  MoveL 11412 to (239.47, 155.25, 153.89) mm, rotated rx 180 ry 0 rz -180 deg; joints [-62.893, 69.046, -92.108, 64.781, 100.282, 20.756]
  MoveL 11413 to (239.47, 155.25, 153.89) mm, rotated rx 180 ry 0 rz -180 deg; joints [-62.893, 69.046, -92.108, 64.781, 100.282, 20.756]
  Call Extruder(262.89466)
  MoveL 11414 to (239.41, 155.44, 153.89) mm, rotated rx 180 ry 0 rz -180 deg; joints [-62.939, 69.059, -92.103, 64.822, 100.258, 20.747]
  MoveL 11415 to (239.41, 155.44, 153.89) mm, rotated rx 180 ry 0 rz -180 deg; joints [-62.939, 69.059, -92.103, 64.822, 100.258, 20.747]
  Call Extruder(263.07662)
  MoveL 11416 to (239.29, 155.73, 153.89) mm, rotated rx 180 ry 0 rz 180 deg; joints [-63.018, 69.079, -92.095, 64.892, 100.218, 20.735]
  MoveL 11417 to (239.29, 155.73, 153.89) mm, rotated rx 180 ry 0 rz 180 deg; joints [-63.018, 69.079, -92.095, 64.892, 100.218, 20.735]
  Call Extruder(263.25933)
  MoveL 11418 to (239.17, 156.02, 153.89) mm, rotated rx 180 ry 0 rz 180 deg; joints [-63.097, 69.098, -92.087, 64.963, 100.179, 20.723]
  MoveL 11419 to (239.17, 156.02, 153.89) mm, rotated rx 180 ry 0 rz 180 deg; joints [-63.097, 69.098, -92.087, 64.963, 100.179, 20.723]
  Call Extruder(263.42975)
  MoveL 11420 to (239.05, 156.29, 153.89) mm, rotated rx 180 ry 0 rz 180 deg; joints [-63.17, 69.116, -92.079, 65.028, 100.142, 20.712]
  MoveL 11421 to (239.05, 156.29, 153.89) mm, rotated rx 180 ry 0 rz 180 deg; joints [-63.17, 69.116, -92.079, 65.028, 100.142, 20.712]
  Call Extruder(263.58776)
  MoveL 11422 to (238.94, 156.54, 153.89) mm, rotated rx 180 ry 0 rz 180 deg; joints [-63.238, 69.132, -92.073, 65.089, 100.108, 20.702]
  MoveL 11423 to (238.94, 156.54, 153.89) mm, rotated rx 180 ry 0 rz 180 deg; joints [-63.238, 69.132, -92.073, 65.089, 100.108, 20.702]
  Call Extruder(263.74638)
  MoveL 11424 to (238.84, 156.79, 153.89) mm, rotated rx 180 ry 0 rz -180 deg; joints [-63.306, 69.149, -92.066, 65.15, 100.074, 20.692]
  MoveL 11425 to (238.84, 156.79, 153.89) mm, rotated rx 180 ry 0 rz -180 deg; joints [-63.306, 69.149, -92.066, 65.15, 100.074, 20.692]
  Call Extruder(263.95255)
  MoveL 11426 to (238.66, 157.09, 153.89) mm, rotated rx 180 ry 0 rz 180 deg; joints [-63.401, 69.167, -92.058, 65.236, 100.03, 20.684]
  MoveL 11427 to (238.66, 157.09, 153.89) mm, rotated rx 180 ry 0 rz 180 deg; joints [-63.401, 69.167, -92.058, 65.236, 100.03, 20.684]
  Call Extruder(264.15949)
  MoveL 11428 to (238.49, 157.4, 153.89) mm, rotated rx 180 ry 0 rz 180 deg; joints [-63.497, 69.185, -92.05, 65.323, 99.985, 20.676]
  MoveL 11429 to (238.49, 157.4, 153.89) mm, rotated rx 180 ry 0 rz 180 deg; joints [-63.497, 69.185, -92.05, 65.323, 99.985, 20.676]
  Call Extruder(264.36722)
  MoveL 11430 to (238.31, 157.7, 153.89) mm, rotated rx 180 ry 0 rz 180 deg; joints [-63.592, 69.203, -92.043, 65.409, 99.941, 20.668]
  MoveL 11431 to (238.31, 157.7, 153.89) mm, rotated rx 180 ry 0 rz 180 deg; joints [-63.592, 69.203, -92.043, 65.409, 99.941, 20.668]
  Call Extruder(264.57572)
  MoveL 11432 to (238.14, 158.01, 153.89) mm, rotated rx 180 ry 0 rz 180 deg; joints [-63.687, 69.222, -92.035, 65.495, 99.897, 20.659]
  MoveL 11433 to (238.14, 158.01, 153.89) mm, rotated rx 180 ry 0 rz 180 deg; joints [-63.687, 69.222, -92.035, 65.495, 99.897, 20.659]
  Call Extruder(264.75269)
  MoveL 11434 to (237.96, 158.25, 153.89) mm, rotated rx -180 ry 0 rz -180 deg; joints [-63.772, 69.235, -92.03, 65.573, 99.859, 20.656]
  MoveL 11435 to (237.96, 158.25, 153.89) mm, rotated rx -180 ry 0 rz -180 deg; joints [-63.772, 69.235, -92.03, 65.573, 99.859, 20.656]
  Call Extruder(265.08090)
  MoveL 11436 to (237.64, 158.69, 153.89) mm, rotated rx 180 ry 0 rz -180 deg; joints [-63.93, 69.259, -92.019, 65.718, 99.789, 20.65]
  MoveL 11437 to (237.64, 158.69, 153.89) mm, rotated rx 180 ry 0 rz -180 deg; joints [-63.93, 69.259, -92.019, 65.718, 99.789, 20.65]
  Call Extruder(265.41030)
  MoveL 11438 to (237.32, 159.14, 153.89) mm, rotated rx 180 ry 0 rz 180 deg; joints [-64.087, 69.283, -92.009, 65.861, 99.72, 20.643]
  Call Extruder(266.28192)
  MoveL 11439 to (236.35, 160.23, 153.89) mm, rotated rx -180 ry 0 rz 180 deg; joints [-64.521, 69.336, -91.987, 66.261, 99.536, 20.642]
  Call Extruder(267.07895)
  MoveL 11440 to (235.35, 161.1, 153.89) mm, rotated rx 180 ry 0 rz -180 deg; joints [-64.933, 69.37, -91.972, 66.645, 99.371, 20.661]
  Call Extruder(267.24365)
  MoveL 11441 to (235.13, 161.27, 153.89) mm, rotated rx 180 ry 0 rz -180 deg; joints [-65.02, 69.375, -91.97, 66.726, 99.338, 20.668]
  MoveL 11442 to (235.13, 161.27, 153.89) mm, rotated rx 180 ry 0 rz -180 deg; joints [-65.02, 69.375, -91.97, 66.726, 99.338, 20.668]
  Call Extruder(267.57190)
  MoveL 11443 to (234.69, 161.59, 153.89) mm, rotated rx -180 ry 0 rz -180 deg; joints [-65.193, 69.385, -91.965, 66.888, 99.271, 20.681]
  MoveL 11444 to (234.69, 161.59, 153.89) mm, rotated rx -180 ry 0 rz -180 deg; joints [-65.193, 69.385, -91.965, 66.888, 99.271, 20.681]
  Call Extruder(267.89900)
  MoveL 11445 to (234.24, 161.91, 153.89) mm, rotated rx 180 ry 0 rz 180 deg; joints [-65.367, 69.395, -91.961, 67.051, 99.204, 20.694]
  MoveL 11446 to (234.24, 161.91, 153.89) mm, rotated rx 180 ry 0 rz 180 deg; joints [-65.367, 69.395, -91.961, 67.051, 99.204, 20.694]
  Call Extruder(268.03352)
  MoveL 11447 to (234.05, 162.02, 153.89) mm, rotated rx 180 ry 0 rz 180 deg; joints [-65.439, 69.397, -91.96, 67.119, 99.177, 20.702]
  MoveL 11448 to (234.05, 162.02, 153.89) mm, rotated rx 180 ry 0 rz 180 deg; joints [-65.439, 69.397, -91.96, 67.119, 99.177, 20.702]
  Call Extruder(268.24883)
  MoveL 11449 to (233.73, 162.21, 153.89) mm, rotated rx -180 ry 0 rz 180 deg; joints [-65.556, 69.4, -91.959, 67.229, 99.134, 20.716]
  MoveL 11450 to (233.73, 162.21, 153.89) mm, rotated rx -180 ry 0 rz 180 deg; joints [-65.556, 69.4, -91.959, 67.229, 99.134, 20.716]
  Call Extruder(268.46330)
  MoveL 11451 to (233.41, 162.39, 153.89) mm, rotated rx 180 ry 0 rz 180 deg; joints [-65.672, 69.403, -91.957, 67.338, 99.091, 20.729]
  MoveL 11452 to (233.41, 162.39, 153.89) mm, rotated rx 180 ry 0 rz 180 deg; joints [-65.672, 69.403, -91.957, 67.338, 99.091, 20.729]
  Call Extruder(268.67694)
  MoveL 11453 to (233.1, 162.57, 153.89) mm, rotated rx -180 ry 0 rz 180 deg; joints [-65.789, 69.407, -91.956, 67.448, 99.048, 20.742]
  MoveL 11454 to (233.1, 162.57, 153.89) mm, rotated rx -180 ry 0 rz 180 deg; joints [-65.789, 69.407, -91.956, 67.448, 99.048, 20.742]
  Call Extruder(268.85614)
  MoveL 11455 to (232.83, 162.71, 153.89) mm, rotated rx 180 ry 0 rz 180 deg; joints [-65.887, 69.408, -91.955, 67.541, 99.013, 20.754]
  MoveL 11456 to (232.83, 162.71, 153.89) mm, rotated rx 180 ry 0 rz 180 deg; joints [-65.887, 69.408, -91.955, 67.541, 99.013, 20.754]
  Call Extruder(269.00184)
  MoveL 11457 to (232.6, 162.81, 153.89) mm, rotated rx 180 ry 0 rz -180 deg; joints [-65.967, 69.408, -91.956, 67.617, 98.984, 20.767]
  MoveL 11458 to (232.6, 162.81, 153.89) mm, rotated rx 180 ry 0 rz -180 deg; joints [-65.967, 69.408, -91.956, 67.617, 98.984, 20.767]
  Call Extruder(269.14703)
  MoveL 11459 to (232.37, 162.91, 153.89) mm, rotated rx 180 ry 0 rz 180 deg; joints [-66.048, 69.407, -91.956, 67.693, 98.956, 20.779]
  MoveL 11460 to (232.37, 162.91, 153.89) mm, rotated rx 180 ry 0 rz 180 deg; joints [-66.048, 69.407, -91.956, 67.693, 98.956, 20.779]
  Call Extruder(269.32977)
  MoveL 11461 to (232.07, 163.03, 153.89) mm, rotated rx 180 ry 0 rz -180 deg; joints [-66.149, 69.407, -91.956, 67.789, 98.92, 20.795]
  MoveL 11462 to (232.07, 163.03, 153.89) mm, rotated rx 180 ry 0 rz -180 deg; joints [-66.149, 69.407, -91.956, 67.789, 98.92, 20.795]
  Call Extruder(269.51175)
  MoveL 11463 to (231.78, 163.15, 153.89) mm, rotated rx -180 ry 0 rz 180 deg; joints [-66.251, 69.406, -91.956, 67.886, 98.885, 20.811]
  MoveL 11464 to (231.78, 163.15, 153.89) mm, rotated rx -180 ry 0 rz 180 deg; joints [-66.251, 69.406, -91.956, 67.886, 98.885, 20.811]
  Call Extruder(269.65909)
  MoveL 11465 to (231.54, 163.24, 153.89) mm, rotated rx 180 ry 0 rz -180 deg; joints [-66.333, 69.405, -91.957, 67.964, 98.856, 20.825]
  MoveL 11466 to (231.54, 163.24, 153.89) mm, rotated rx 180 ry 0 rz -180 deg; joints [-66.333, 69.405, -91.957, 67.964, 98.856, 20.825]
  Call Extruder(269.77231)
  MoveL 11467 to (231.35, 163.3, 153.89) mm, rotated rx 180 ry 0 rz -180 deg; joints [-66.397, 69.403, -91.958, 68.024, 98.834, 20.836]
  MoveL 11468 to (231.35, 163.3, 153.89) mm, rotated rx 180 ry 0 rz -180 deg; joints [-66.397, 69.403, -91.958, 68.024, 98.834, 20.836]
  Call Extruder(269.88509)
  MoveL 11469 to (231.17, 163.36, 153.89) mm, rotated rx 180 ry 0 rz 180 deg; joints [-66.46, 69.401, -91.958, 68.085, 98.813, 20.848]
  MoveL 11470 to (231.17, 163.36, 153.89) mm, rotated rx 180 ry 0 rz 180 deg; joints [-66.46, 69.401, -91.958, 68.085, 98.813, 20.848]
  Call Extruder(269.99742)
  MoveL 11471 to (230.98, 163.42, 153.89) mm, rotated rx -180 ry 0 rz -180 deg; joints [-66.524, 69.399, -91.959, 68.145, 98.791, 20.859]
  MoveL 11472 to (230.98, 163.42, 153.89) mm, rotated rx -180 ry 0 rz -180 deg; joints [-66.524, 69.399, -91.959, 68.145, 98.791, 20.859]
  Call Extruder(270.10931)
  MoveL 11473 to (230.79, 163.48, 153.89) mm, rotated rx -180 ry 0 rz 180 deg; joints [-66.587, 69.398, -91.96, 68.205, 98.77, 20.871]
  MoveL 11474 to (230.79, 163.48, 153.89) mm, rotated rx -180 ry 0 rz 180 deg; joints [-66.587, 69.398, -91.96, 68.205, 98.77, 20.871]
  Call Extruder(270.23072)
  MoveL 11475 to (230.58, 163.55, 153.89) mm, rotated rx 180 ry 0 rz -180 deg; joints [-66.656, 69.395, -91.961, 68.271, 98.746, 20.884]
  MoveL 11476 to (230.58, 163.55, 153.89) mm, rotated rx 180 ry 0 rz -180 deg; joints [-66.656, 69.395, -91.961, 68.271, 98.746, 20.884]
  Call Extruder(270.36153)
  MoveL 11477 to (230.36, 163.62, 153.89) mm, rotated rx -180 ry 0 rz 180 deg; joints [-66.731, 69.393, -91.962, 68.342, 98.721, 20.898]
  MoveL 11478 to (230.36, 163.62, 153.89) mm, rotated rx -180 ry 0 rz 180 deg; joints [-66.731, 69.393, -91.962, 68.342, 98.721, 20.898]
  Call Extruder(270.49178)
  MoveL 11479 to (230.14, 163.68, 153.89) mm, rotated rx 180 ry 0 rz -180 deg; joints [-66.805, 69.391, -91.963, 68.413, 98.695, 20.912]
  MoveL 11480 to (230.14, 163.68, 153.89) mm, rotated rx 180 ry 0 rz -180 deg; joints [-66.805, 69.391, -91.963, 68.413, 98.695, 20.912]
  Call Extruder(270.62146)
  MoveL 11481 to (229.91, 163.75, 153.89) mm, rotated rx 180 ry 0 rz 180 deg; joints [-66.88, 69.388, -91.964, 68.484, 98.67, 20.926]
  MoveL 11482 to (229.91, 163.75, 153.89) mm, rotated rx 180 ry 0 rz 180 deg; joints [-66.88, 69.388, -91.964, 68.484, 98.67, 20.926]
  Call Extruder(270.75058)
  MoveL 11483 to (229.69, 163.82, 153.89) mm, rotated rx 180 ry 0 rz -180 deg; joints [-66.955, 69.386, -91.965, 68.555, 98.645, 20.939]
  MoveL 11484 to (229.69, 163.82, 153.89) mm, rotated rx 180 ry 0 rz -180 deg; joints [-66.955, 69.386, -91.965, 68.555, 98.645, 20.939]
  Call Extruder(270.86565)
  MoveL 11485 to (229.48, 163.86, 153.89) mm, rotated rx 180 ry 0 rz 180 deg; joints [-67.021, 69.382, -91.967, 68.619, 98.623, 20.954]
  MoveL 11486 to (229.48, 163.86, 153.89) mm, rotated rx 180 ry 0 rz 180 deg; joints [-67.021, 69.382, -91.967, 68.619, 98.623, 20.954]
  Call Extruder(270.98027)
  MoveL 11487 to (229.28, 163.91, 153.89) mm, rotated rx 180 ry 0 rz 180 deg; joints [-67.087, 69.379, -91.968, 68.682, 98.601, 20.968]
  MoveL 11488 to (229.28, 163.91, 153.89) mm, rotated rx 180 ry 0 rz 180 deg; joints [-67.087, 69.379, -91.968, 68.682, 98.601, 20.968]
  Call Extruder(271.09444)
  MoveL 11489 to (229.08, 163.95, 153.89) mm, rotated rx 180 ry 0 rz 180 deg; joints [-67.153, 69.375, -91.97, 68.745, 98.579, 20.982]
  MoveL 11490 to (229.08, 163.95, 153.89) mm, rotated rx 180 ry 0 rz 180 deg; joints [-67.153, 69.375, -91.97, 68.745, 98.579, 20.982]
  Call Extruder(271.20816)
  MoveL 11491 to (228.87, 164, 153.89) mm, rotated rx -180 ry 0 rz -180 deg; joints [-67.22, 69.371, -91.971, 68.808, 98.557, 20.996]
  MoveL 11492 to (228.87, 164, 153.89) mm, rotated rx -180 ry 0 rz -180 deg; joints [-67.22, 69.371, -91.971, 68.808, 98.557, 20.996]
  Call Extruder(271.33358)
  MoveL 11493 to (228.65, 164.04, 153.89) mm, rotated rx 180 ry 0 rz -180 deg; joints [-67.293, 69.367, -91.973, 68.878, 98.533, 21.012]
  MoveL 11494 to (228.65, 164.04, 153.89) mm, rotated rx 180 ry 0 rz -180 deg; joints [-67.293, 69.367, -91.973, 68.878, 98.533, 21.012]
  Call Extruder(271.47056)
  MoveL 11495 to (228.4, 164.09, 153.89) mm, rotated rx -180 ry 0 rz 180 deg; joints [-67.373, 69.363, -91.975, 68.955, 98.507, 21.029]
  MoveL 11496 to (228.4, 164.09, 153.89) mm, rotated rx -180 ry 0 rz 180 deg; joints [-67.373, 69.363, -91.975, 68.955, 98.507, 21.029]
  Call Extruder(271.60692)
  MoveL 11497 to (228.15, 164.14, 153.89) mm, rotated rx 180 ry 0 rz 180 deg; joints [-67.453, 69.358, -91.977, 69.032, 98.48, 21.047]
  MoveL 11498 to (228.15, 164.14, 153.89) mm, rotated rx 180 ry 0 rz 180 deg; joints [-67.453, 69.358, -91.977, 69.032, 98.48, 21.047]
  Call Extruder(271.74268)
  MoveL 11499 to (227.9, 164.19, 153.89) mm, rotated rx 180 ry 0 rz 180 deg; joints [-67.534, 69.353, -91.979, 69.108, 98.454, 21.064]
  MoveL 11500 to (227.9, 164.19, 153.89) mm, rotated rx 180 ry 0 rz 180 deg; joints [-67.534, 69.353, -91.979, 69.108, 98.454, 21.064]
  Call Extruder(271.87783)
  MoveL 11501 to (227.65, 164.24, 153.89) mm, rotated rx 180 ry 0 rz -180 deg; joints [-67.614, 69.349, -91.981, 69.185, 98.427, 21.082]
  MoveL 11502 to (227.65, 164.24, 153.89) mm, rotated rx 180 ry 0 rz -180 deg; joints [-67.614, 69.349, -91.981, 69.185, 98.427, 21.082]
  Call Extruder(272.01237)
  MoveL 11503 to (227.4, 164.29, 153.89) mm, rotated rx 180 ry 0 rz 180 deg; joints [-67.695, 69.344, -91.983, 69.262, 98.401, 21.099]
  MoveL 11504 to (227.4, 164.29, 153.89) mm, rotated rx 180 ry 0 rz 180 deg; joints [-67.695, 69.344, -91.983, 69.262, 98.401, 21.099]
  Call Extruder(272.14629)
  MoveL 11505 to (227.15, 164.34, 153.89) mm, rotated rx -180 ry 0 rz -180 deg; joints [-67.775, 69.34, -91.985, 69.338, 98.374, 21.116]
  MoveL 11506 to (227.15, 164.34, 153.89) mm, rotated rx -180 ry 0 rz -180 deg; joints [-67.775, 69.34, -91.985, 69.338, 98.374, 21.116]
  Call Extruder(272.29416)
  MoveL 11507 to (226.87, 164.39, 153.89) mm, rotated rx 180 ry 0 rz 180 deg; joints [-67.864, 69.334, -91.987, 69.423, 98.345, 21.136]
  MoveL 11508 to (226.87, 164.39, 153.89) mm, rotated rx 180 ry 0 rz 180 deg; joints [-67.864, 69.334, -91.987, 69.423, 98.345, 21.136]
  Call Extruder(272.45590)
  MoveL 11509 to (226.57, 164.44, 153.89) mm, rotated rx -180 ry 0 rz -180 deg; joints [-67.961, 69.328, -91.99, 69.516, 98.313, 21.158]
  MoveL 11510 to (226.57, 164.44, 153.89) mm, rotated rx -180 ry 0 rz -180 deg; joints [-67.961, 69.328, -91.99, 69.516, 98.313, 21.158]
  Call Extruder(272.61691)
  MoveL 11511 to (226.26, 164.49, 153.89) mm, rotated rx 180 ry 0 rz 180 deg; joints [-68.059, 69.321, -91.993, 69.609, 98.281, 21.18]
  MoveL 11512 to (226.26, 164.49, 153.89) mm, rotated rx 180 ry 0 rz 180 deg; joints [-68.059, 69.321, -91.993, 69.609, 98.281, 21.18]
  Call Extruder(272.77720)
  MoveL 11513 to (225.96, 164.54, 153.89) mm, rotated rx 180 ry 0 rz -180 deg; joints [-68.156, 69.315, -91.996, 69.703, 98.249, 21.202]
  MoveL 11514 to (225.96, 164.54, 153.89) mm, rotated rx 180 ry 0 rz -180 deg; joints [-68.156, 69.315, -91.996, 69.703, 98.249, 21.202]
  Call Extruder(272.93675)
  MoveL 11515 to (225.65, 164.58, 153.89) mm, rotated rx 180 ry 0 rz -180 deg; joints [-68.254, 69.308, -91.998, 69.796, 98.217, 21.224]
  MoveL 11516 to (225.65, 164.58, 153.89) mm, rotated rx 180 ry 0 rz -180 deg; joints [-68.254, 69.308, -91.998, 69.796, 98.217, 21.224]
  Call Extruder(273.09558)
  MoveL 11517 to (225.34, 164.63, 153.89) mm, rotated rx 180 ry 0 rz 180 deg; joints [-68.351, 69.302, -92.001, 69.889, 98.184, 21.245]
  MoveL 11518 to (225.34, 164.63, 153.89) mm, rotated rx 180 ry 0 rz 180 deg; joints [-68.351, 69.302, -92.001, 69.889, 98.184, 21.245]
  Call Extruder(273.27425)
  MoveL 11519 to (225, 164.68, 153.89) mm, rotated rx 180 ry 0 rz -180 deg; joints [-68.461, 69.294, -92.004, 69.994, 98.148, 21.271]
  MoveL 11520 to (225, 164.68, 153.89) mm, rotated rx 180 ry 0 rz -180 deg; joints [-68.461, 69.294, -92.004, 69.994, 98.148, 21.271]
  Call Extruder(273.47269)
  MoveL 11521 to (224.61, 164.73, 153.89) mm, rotated rx -180 ry 0 rz -180 deg; joints [-68.583, 69.285, -92.008, 70.111, 98.109, 21.3]
  MoveL 11522 to (224.61, 164.73, 153.89) mm, rotated rx -180 ry 0 rz -180 deg; joints [-68.583, 69.285, -92.008, 70.111, 98.109, 21.3]
  Call Extruder(273.67027)
  MoveL 11523 to (224.22, 164.77, 153.89) mm, rotated rx 180 ry 0 rz 180 deg; joints [-68.706, 69.276, -92.012, 70.228, 98.069, 21.328]
  MoveL 11524 to (224.22, 164.77, 153.89) mm, rotated rx 180 ry 0 rz 180 deg; joints [-68.706, 69.276, -92.012, 70.228, 98.069, 21.328]
  Call Extruder(273.86697)
  MoveL 11525 to (223.84, 164.82, 153.89) mm, rotated rx 180 ry 0 rz 180 deg; joints [-68.828, 69.266, -92.016, 70.344, 98.028, 21.357]
  MoveL 11526 to (223.84, 164.82, 153.89) mm, rotated rx 180 ry 0 rz 180 deg; joints [-68.828, 69.266, -92.016, 70.344, 98.028, 21.357]
  Call Extruder(274.06281)
  MoveL 11527 to (223.45, 164.86, 153.89) mm, rotated rx 180 ry 0 rz 180 deg; joints [-68.951, 69.257, -92.02, 70.461, 97.988, 21.385]
  MoveL 11528 to (223.45, 164.86, 153.89) mm, rotated rx 180 ry 0 rz 180 deg; joints [-68.951, 69.257, -92.02, 70.461, 97.988, 21.385]
  Call Extruder(274.35817)
  MoveL 11529 to (222.86, 164.91, 153.89) mm, rotated rx 180 ry 0 rz 180 deg; joints [-69.135, 69.242, -92.027, 70.637, 97.928, 21.43]
  MoveL 11530 to (222.86, 164.91, 153.89) mm, rotated rx 180 ry 0 rz 180 deg; joints [-69.135, 69.242, -92.027, 70.637, 97.928, 21.43]
  Call Extruder(274.65220)
  MoveL 11531 to (222.27, 164.96, 153.89) mm, rotated rx 180 ry 0 rz 180 deg; joints [-69.319, 69.226, -92.033, 70.813, 97.868, 21.475]
  MoveL 11532 to (222.27, 164.96, 153.89) mm, rotated rx 180 ry 0 rz 180 deg; joints [-69.319, 69.226, -92.033, 70.813, 97.868, 21.475]
  Call Extruder(274.94489)
  MoveL 11533 to (221.68, 165, 153.89) mm, rotated rx 180 ry 0 rz 180 deg; joints [-69.504, 69.211, -92.04, 70.99, 97.808, 21.52]
  MoveL 11534 to (221.68, 165, 153.89) mm, rotated rx 180 ry 0 rz 180 deg; joints [-69.504, 69.211, -92.04, 70.99, 97.808, 21.52]
  Call Extruder(275.51834)
  MoveL 11535 to (220.52, 165.05, 153.89) mm, rotated rx 180 ry 0 rz 180 deg; joints [-69.864, 69.177, -92.054, 71.334, 97.691, 21.611]
  MoveL 11536 to (220.52, 165.05, 153.89) mm, rotated rx 180 ry 0 rz 180 deg; joints [-69.864, 69.177, -92.054, 71.334, 97.691, 21.611]
  Call Extruder(276.23235)
  MoveL 11537 to (219.06, 165.09, 153.89) mm, rotated rx 180 ry 0 rz 180 deg; joints [-70.315, 69.134, -92.072, 71.764, 97.544, 21.726]
  Call Extruder(393.07903)
  MoveL 11538 to (-19.06, 165.09, 153.89) mm, rotated rx -180 ry 0 rz 180 deg; joints [-137.325, 74.771, -88.513, 136.495, 79.942, 9.412]
  Call Extruder(393.50763)
  MoveL 11539 to (-19.94, 165.07, 153.89) mm, rotated rx -180 ry 0 rz 180 deg; joints [-137.467, 74.815, -88.471, 136.648, 79.981, 9.327]
  MoveL 11540 to (-19.94, 165.07, 153.89) mm, rotated rx -180 ry 0 rz 180 deg; joints [-137.467, 74.815, -88.471, 136.648, 79.981, 9.327]
  Call Extruder(394.08108)
  MoveL 11541 to (-21.1, 165.03, 153.89) mm, rotated rx 180 ry 0 rz -180 deg; joints [-137.659, 74.874, -88.417, 136.853, 80.032, 9.216]
  MoveL 11542 to (-21.1, 165.03, 153.89) mm, rotated rx 180 ry 0 rz -180 deg; joints [-137.659, 74.874, -88.417, 136.853, 80.032, 9.216]
  Call Extruder(394.51538)
  MoveL 11543 to (-21.97, 164.98, 153.89) mm, rotated rx -180 ry 0 rz -180 deg; joints [-137.804, 74.917, -88.377, 137.009, 80.07, 9.133]
  MoveL 11544 to (-21.97, 164.98, 153.89) mm, rotated rx -180 ry 0 rz -180 deg; joints [-137.804, 74.917, -88.377, 137.009, 80.07, 9.133]
  Call Extruder(394.80941)
  MoveL 11545 to (-22.56, 164.93, 153.89) mm, rotated rx 180 ry 0 rz 180 deg; joints [-137.905, 74.945, -88.35, 137.116, 80.094, 9.077]
  MoveL 11546 to (-22.56, 164.93, 153.89) mm, rotated rx 180 ry 0 rz 180 deg; joints [-137.905, 74.945, -88.35, 137.116, 80.094, 9.077]
  Call Extruder(395.10477)
  MoveL 11547 to (-23.15, 164.89, 153.89) mm, rotated rx 180 ry 0 rz 180 deg; joints [-138.004, 74.974, -88.323, 137.223, 80.119, 9.022]
  MoveL 11548 to (-23.15, 164.89, 153.89) mm, rotated rx 180 ry 0 rz 180 deg; joints [-138.004, 74.974, -88.323, 137.223, 80.119, 9.022]
  Call Extruder(395.35098)
  MoveL 11549 to (-23.64, 164.84, 153.89) mm, rotated rx -180 ry 0 rz -180 deg; joints [-138.088, 74.997, -88.301, 137.312, 80.139, 8.976]
  MoveL 11550 to (-23.64, 164.84, 153.89) mm, rotated rx -180 ry 0 rz -180 deg; joints [-138.088, 74.997, -88.301, 137.312, 80.139, 8.976]
  Call Extruder(395.54769)
  MoveL 11551 to (-24.03, 164.79, 153.89) mm, rotated rx 180 ry 0 rz -180 deg; joints [-138.156, 75.015, -88.284, 137.385, 80.154, 8.941]
  MoveL 11552 to (-24.03, 164.79, 153.89) mm, rotated rx 180 ry 0 rz -180 deg; joints [-138.156, 75.015, -88.284, 137.385, 80.154, 8.941]
  Call Extruder(395.74526)
  MoveL 11553 to (-24.42, 164.75, 153.89) mm, rotated rx -180 ry 0 rz 180 deg; joints [-138.224, 75.033, -88.267, 137.457, 80.17, 8.905]
  MoveL 11554 to (-24.42, 164.75, 153.89) mm, rotated rx -180 ry 0 rz 180 deg; joints [-138.224, 75.033, -88.267, 137.457, 80.17, 8.905]
  Call Extruder(395.94370)
  MoveL 11555 to (-24.8, 164.7, 153.89) mm, rotated rx 180 ry 0 rz 180 deg; joints [-138.292, 75.051, -88.25, 137.529, 80.185, 8.869]
  MoveL 11556 to (-24.8, 164.7, 153.89) mm, rotated rx 180 ry 0 rz 180 deg; joints [-138.292, 75.051, -88.25, 137.529, 80.185, 8.869]
  Call Extruder(396.14301)
  MoveL 11557 to (-25.19, 164.66, 153.89) mm, rotated rx -180 ry 0 rz 180 deg; joints [-138.359, 75.069, -88.233, 137.6, 80.201, 8.834]
  MoveL 11558 to (-25.19, 164.66, 153.89) mm, rotated rx -180 ry 0 rz 180 deg; joints [-138.359, 75.069, -88.233, 137.6, 80.201, 8.834]
  Call Extruder(396.30184)
  MoveL 11559 to (-25.5, 164.61, 153.89) mm, rotated rx 180 ry 0 rz -180 deg; joints [-138.415, 75.082, -88.22, 137.659, 80.212, 8.806]
  MoveL 11560 to (-25.5, 164.61, 153.89) mm, rotated rx 180 ry 0 rz -180 deg; joints [-138.415, 75.082, -88.22, 137.659, 80.212, 8.806]
  Call Extruder(396.46140)
  MoveL 11561 to (-25.8, 164.56, 153.89) mm, rotated rx -180 ry 0 rz 180 deg; joints [-138.47, 75.096, -88.207, 137.718, 80.223, 8.778]
  MoveL 11562 to (-25.8, 164.56, 153.89) mm, rotated rx -180 ry 0 rz 180 deg; joints [-138.47, 75.096, -88.207, 137.718, 80.223, 8.778]
  Call Extruder(396.62169)
  MoveL 11563 to (-26.11, 164.51, 153.89) mm, rotated rx 180 ry 0 rz 180 deg; joints [-138.525, 75.109, -88.193, 137.776, 80.235, 8.751]
  MoveL 11564 to (-26.11, 164.51, 153.89) mm, rotated rx 180 ry 0 rz 180 deg; joints [-138.525, 75.109, -88.193, 137.776, 80.235, 8.751]
  Call Extruder(396.78271)
  MoveL 11565 to (-26.41, 164.46, 153.89) mm, rotated rx 180 ry 0 rz 180 deg; joints [-138.58, 75.123, -88.18, 137.834, 80.246, 8.723]
  MoveL 11566 to (-26.41, 164.46, 153.89) mm, rotated rx 180 ry 0 rz 180 deg; joints [-138.58, 75.123, -88.18, 137.834, 80.246, 8.723]
  Call Extruder(396.94445)
  MoveL 11567 to (-26.72, 164.41, 153.89) mm, rotated rx -180 ry 0 rz 180 deg; joints [-138.635, 75.137, -88.167, 137.892, 80.258, 8.695]
  MoveL 11568 to (-26.72, 164.41, 153.89) mm, rotated rx -180 ry 0 rz 180 deg; joints [-138.635, 75.137, -88.167, 137.892, 80.258, 8.695]
  Call Extruder(397.10692)
  MoveL 11569 to (-27.03, 164.36, 153.89) mm, rotated rx 180 ry 0 rz 180 deg; joints [-138.69, 75.15, -88.154, 137.95, 80.269, 8.668]
  MoveL 11570 to (-27.03, 164.36, 153.89) mm, rotated rx 180 ry 0 rz 180 deg; joints [-138.69, 75.15, -88.154, 137.95, 80.269, 8.668]
  Call Extruder(397.24085)
  MoveL 11571 to (-27.27, 164.32, 153.89) mm, rotated rx -180 ry 0 rz 180 deg; joints [-138.736, 75.161, -88.144, 137.999, 80.278, 8.646]
  MoveL 11572 to (-27.27, 164.32, 153.89) mm, rotated rx -180 ry 0 rz 180 deg; joints [-138.736, 75.161, -88.144, 137.999, 80.278, 8.646]
  Call Extruder(397.37538)
  MoveL 11573 to (-27.52, 164.27, 153.89) mm, rotated rx 180 ry 0 rz 180 deg; joints [-138.783, 75.172, -88.133, 138.048, 80.287, 8.624]
  MoveL 11574 to (-27.52, 164.27, 153.89) mm, rotated rx 180 ry 0 rz 180 deg; joints [-138.783, 75.172, -88.133, 138.048, 80.287, 8.624]
  Call Extruder(397.51053)
  MoveL 11575 to (-27.77, 164.22, 153.89) mm, rotated rx 180 ry 0 rz 180 deg; joints [-138.829, 75.182, -88.123, 138.097, 80.295, 8.602]
  MoveL 11576 to (-27.77, 164.22, 153.89) mm, rotated rx 180 ry 0 rz 180 deg; joints [-138.829, 75.182, -88.123, 138.097, 80.295, 8.602]
  Call Extruder(397.64629)
  MoveL 11577 to (-28.02, 164.17, 153.89) mm, rotated rx -180 ry 0 rz 180 deg; joints [-138.875, 75.193, -88.112, 138.146, 80.304, 8.58]
  MoveL 11578 to (-28.02, 164.17, 153.89) mm, rotated rx -180 ry 0 rz 180 deg; joints [-138.875, 75.193, -88.112, 138.146, 80.304, 8.58]
  Call Extruder(397.78265)
  MoveL 11579 to (-28.27, 164.12, 153.89) mm, rotated rx 180 ry 0 rz 180 deg; joints [-138.921, 75.203, -88.102, 138.195, 80.313, 8.558]
  MoveL 11580 to (-28.27, 164.12, 153.89) mm, rotated rx 180 ry 0 rz 180 deg; joints [-138.921, 75.203, -88.102, 138.195, 80.313, 8.558]
  Call Extruder(397.86751)
  MoveL 11581 to (-28.43, 164.09, 153.89) mm, rotated rx 180 ry 0 rz 180 deg; joints [-138.95, 75.21, -88.095, 138.225, 80.318, 8.544]
  Set speed (130.0 mm/s)
  MoveL 11582 to (-31.76, 163.31, 153.89) mm, rotated rx -180 ry 0 rz 180 deg; joints [-139.581, 75.348, -87.959, 138.889, 80.432, 8.254]
  Call Extruder(395.86751)
  Set speed (40.0 mm/s)
  MoveL 11583 to (-31.76, 163.31, 153.89) mm, rotated rx -180 ry 0 rz 180 deg; joints [-139.581, 75.348, -87.959, 138.889, 80.432, 8.254]
  Set speed (1000.0 mm/s)
  Call Extruder(-1)
  MoveL 11584 to (-31.76, 163.31, 153.89) mm, rotated rx -180 ry 0 rz 180 deg; joints [-139.581, 75.348, -87.959, 138.889, 80.432, 8.254]
  Call Extruder(0.00000)
  Call M_RunCode(107)
  Call M_RunCode(104)
  Call M_RunCode(84)
  Call M_RunCode(140)

--- program Prog4 (robot Denso VS-6577G-B) ---
  Set Ref.: Ref001
  Set Tool: nozzle
  MoveJ (First 1)
  MoveL (First 2)
  MoveL (First 3)
  MoveL (First 4)
  MoveL (First 1)
  MoveL (Second 1)
  MoveL (Second 2)
  MoveL (Second 3)
  MoveL (Second 4)
  MoveL (Second 1)
  MoveL (Third 1)
  MoveL (Third 2)
  MoveL (Third 3)
  MoveL (Third 4)
  MoveL (Third 1)
  MoveL (Fourth 1)
  MoveL (Fourth 2)
  MoveL (Fourth 3)
  MoveL (Fourth 4)
  MoveL (Fourth 1)
